(* IEC 61131-3 sources: Industry-PLC-LLM/data/PLCBEAD_repo/PLCBEAD_PLCEmbed-main/PLC-BEAD/Source/GEB/_INT_TO_UDINT, 1 file *)

(* ---- _INT_TO_UDINT.ST ---- *)
FUNCTION _INT_TO_UDINT:UDINT
	VAR_INPUT
		IN :	INT;
	END_VAR

	_INT_TO_UDINT := DINT_TO_UDINT(INT_TO_DINT(IN));
END_FUNCTION

PROGRAM program0
  VAR
    LocalVar0 : INT;
	LocalOUT  : UDINT;
  END_VAR

  LocalOUT := _INT_TO_UDINT(LocalVar0);
END_PROGRAM
